LIN {X -0.074,Y -440.123,Z 231.770,A 0.000,B 0.000,C 90.000,E1 153.973} C_DIS
LIN {X 0.244,Y -443.570,Z 231.757,A 0.000,B 0.000,C 90.000,E1 151.307} C_DIS
LIN {X -0.099,Y -447.476,Z 231.744,A 0.000,B 0.000,C 90.000,E1 148.742} C_DIS
LIN {X -0.036,Y -450.606,Z 231.734,A 0.000,B 0.000,C 90.000,E1 146.786} C_DIS
LIN {X -0.031,Y -453.961,Z 231.724,A 0.000,B 0.000,C 90.000,E1 144.848} C_DIS
LIN {X -0.148,Y -456.732,Z 231.716,A 0.000,B 0.000,C 90.000,E1 143.256} C_DIS
LIN {X 0.157,Y -459.197,Z 231.708,A 0.000,B 0.000,C 90.000,E1 141.618} C_DIS
LIN {X -0.219,Y -461.363,Z 231.700,A 0.000,B 0.000,C 90.000,E1 140.070} C_DIS
LIN {X -0.002,Y -462.909,Z 231.694,A 0.000,B 0.000,C 90.000,E1 138.771} C_DIS
LIN {X -0.018,Y -464.342,Z 231.686,A 0.000,B 0.000,C 90.000,E1 137.187} C_DIS
LIN {X 0.219,Y -465.215,Z 231.680,A 0.000,B 0.000,C 90.000,E1 135.891} C_DIS
LIN {X -0.247,Y -465.696,Z 231.675,A 0.000,B 0.000,C 90.000,E1 135.000} C_DIS
LIN {X 0.017,Y -465.978,Z 231.669,A 0.000,B 0.000,C 90.000,E1 133.704} C_DIS
LIN {X -0.105,Y -465.940,Z 231.664,A 0.000,B 0.000,C 90.000,E1 132.771} C_DIS
LIN {X -0.166,Y -465.456,Z 231.657,A 0.000,B 0.000,C 90.000,E1 131.515} C_DIS
LIN {X -0.138,Y -464.609,Z 231.650,A 0.000,B 0.000,C 90.000,E1 129.930} C_DIS
LIN {X 0.071,Y -464.004,Z 231.645,A 0.000,B 0.000,C 90.000,E1 128.955} C_DIS
LIN {X 0.099,Y -462.931,Z 231.639,A 0.000,B 0.000,C 90.000,E1 127.684} C_DIS
LIN {X 0.027,Y -461.600,Z 231.632,A 0.000,B 0.000,C 90.000,E1 126.423} C_DIS
LIN {X 0.014,Y -460.384,Z 231.627,A 0.000,B 0.000,C 90.000,E1 125.471} C_DIS
LIN {X 0.112,Y -458.220,Z 231.619,A 0.000,B 0.000,C 90.000,E1 123.865} C_DIS
LIN {X -0.088,Y -455.689,Z 231.611,A 0.000,B 0.000,C 90.000,E1 122.291} C_DIS
LIN {X -0.055,Y -453.556,Z 231.605,A 0.000,B 0.000,C 90.000,E1 121.003} C_DIS
LIN {X -0.065,Y -451.335,Z 231.599,A 0.000,B 0.000,C 90.000,E1 119.716} C_DIS
LIN {X -0.010,Y -447.845,Z 231.589,A 0.000,B 0.000,C 90.000,E1 117.769} C_DIS
LIN {X -0.234,Y -444.436,Z 231.579,A 0.000,B 0.000,C 90.000,E1 115.848} C_DIS
LIN {X 0.063,Y -443.558,Z 231.577,A 0.000,B 0.000,C 90.000,E1 115.335} C_DIS
LIN {X 0.024,Y -443.550,Z 231.577,A 0.000,B 0.000,C 90.000,E1 115.335} C_DIS
LIN {X -0.070,Y -444.990,Z 231.574,A 0.000,B 0.000,C 90.000,E1 114.847} C_DIS
LIN {X 0.206,Y -454.125,Z 231.555,A 0.000,B 0.000,C 90.000,E1 110.918} C_DIS
LIN {X -0.107,Y -456.781,Z 231.550,A 0.000,B 0.000,C 90.000,E1 109.993} C_DIS
LIN {X 0.225,Y -457.541,Z 231.548,A 0.000,B 0.000,C 90.000,E1 109.631} C_DIS
LIN {X -0.136,Y -466.232,Z 231.528,A 0.000,B 0.000,C 90.000,E1 105.536} C_DIS
LIN {X -0.085,Y -467.792,Z 231.524,A 0.000,B 0.000,C 90.000,E1 104.898} C_DIS
LIN {X -0.114,Y -475.999,Z 231.501,A 0.000,B 0.000,C 90.000,E1 100.197} C_DIS
LIN {X 0.036,Y -476.693,Z 231.498,A 0.000,B 0.000,C 90.000,E1 99.557} C_DIS
LIN {X 0.160,Y -481.938,Z 231.478,A 0.000,B 0.000,C 90.000,E1 95.511} C_DIS
LIN {X 0.008,Y -482.209,Z 231.476,A 0.000,B 0.000,C 90.000,E1 95.220} C_DIS
LIN {X -0.054,Y -485.406,Z 231.455,A 0.000,B 0.000,C 90.000,E1 90.917} C_DIS
LIN {X -0.228,Y -485.528,Z 231.453,A 0.000,B 0.000,C 90.000,E1 90.630} C_DIS
LIN {X -0.021,Y -486.366,Z 231.433,A 0.000,B 0.000,C 90.000,E1 86.617} C_DIS
LIN {X -0.196,Y -486.368,Z 231.432,A 0.000,B 0.000,C 90.000,E1 86.331} C_DIS
LIN {X 0.138,Y -485.674,Z 231.425,A 0.000,B 0.000,C 90.000,E1 85.065} C_DIS
LIN {X -0.172,Y -484.691,Z 231.409,A 0.000,B 0.000,C 90.000,E1 81.724} C_DIS
LIN {X 0.174,Y -484.487,Z 231.407,A 0.000,B 0.000,C 90.000,E1 81.376} C_DIS
LIN {X 0.178,Y -480.662,Z 231.385,A 0.000,B 0.000,C 90.000,E1 77.061} C_DIS
LIN {X 0.144,Y -480.414,Z 231.384,A 0.000,B 0.000,C 90.000,E1 76.756} C_DIS
LIN {X -0.084,Y -474.193,Z 231.361,A 0.000,B 0.000,C 90.000,E1 72.127} C_DIS
LIN {X -0.150,Y -473.017,Z 231.357,A 0.000,B 0.000,C 90.000,E1 71.511} C_DIS
LIN {X -0.050,Y -465.699,Z 231.335,A 0.000,B 0.000,C 90.000,E1 67.102} C_DIS
LIN {X 0.008,Y -459.410,Z 231.321,A 0.000,B 0.000,C 90.000,E1 64.152} C_DIS
LIN {X -0.032,Y -459.417,Z 231.321,A 0.000,B 0.000,C 90.000,E1 64.152} C_DIS
LIN {X -0.197,Y -461.625,Z 231.317,A 0.000,B 0.000,C 90.000,E1 63.384} C_DIS
LIN {X -0.034,Y -464.697,Z 231.312,A 0.000,B 0.000,C 90.000,E1 62.410} C_DIS
LIN {X 0.169,Y -467.308,Z 231.307,A 0.000,B 0.000,C 90.000,E1 61.435} C_DIS
LIN {X -0.164,Y -468.856,Z 231.304,A 0.000,B 0.000,C 90.000,E1 60.845} C_DIS
LIN {X -0.007,Y -469.418,Z 231.303,A 0.000,B 0.000,C 90.000,E1 60.511} C_DIS
LIN {X -0.157,Y -470.244,Z 231.299,A 0.000,B 0.000,C 90.000,E1 59.744} C_DIS
LIN {X 0.008,Y -471.991,Z 231.296,A 0.000,B 0.000,C 90.000,E1 59.253} C_DIS
LIN {X -0.065,Y -473.436,Z 231.295,A 0.000,B 0.000,C 90.000,E1 58.948} C_DIS
LIN {X 0.111,Y -474.609,Z 231.293,A 0.000,B 0.000,C 90.000,E1 58.614} C_DIS
LIN {X 0.070,Y -476.278,Z 231.290,A 0.000,B 0.000,C 90.000,E1 57.995} C_DIS
LIN {X -0.146,Y -477.003,Z 231.288,A 0.000,B 0.000,C 90.000,E1 57.709} C_DIS
LIN {X 0.046,Y -477.537,Z 231.287,A 0.000,B 0.000,C 90.000,E1 57.375} C_DIS
LIN {X 0.007,Y -477.986,Z 231.285,A 0.000,B 0.000,C 90.000,E1 56.914} C_DIS
LIN {X -0.071,Y -480.360,Z 231.281,A 0.000,B 0.000,C 90.000,E1 56.294} C_DIS
LIN {X 0.129,Y -481.734,Z 231.280,A 0.000,B 0.000,C 90.000,E1 55.960} C_DIS
LIN {X -0.063,Y -482.676,Z 231.278,A 0.000,B 0.000,C 90.000,E1 55.674} C_DIS
LIN {X -0.253,Y -483.355,Z 231.277,A 0.000,B 0.000,C 90.000,E1 55.388} C_DIS
LIN {X -0.041,Y -483.816,Z 231.275,A 0.000,B 0.000,C 90.000,E1 55.055} C_DIS
LIN {X -0.223,Y -483.883,Z 231.274,A 0.000,B 0.000,C 90.000,E1 54.769} C_DIS
LIN {X -0.173,Y -483.679,Z 231.273,A 0.000,B 0.000,C 90.000,E1 54.609} C_DIS
LIN {X 0.180,Y -483.698,Z 231.273,A 0.000,B 0.000,C 90.000,E1 54.562} C_DIS
LIN {X 0.272,Y -484.576,Z 231.272,A 0.000,B 0.000,C 90.000,E1 54.402} C_DIS
LIN {X -0.082,Y -486.780,Z 231.269,A 0.000,B 0.000,C 90.000,E1 53.829} C_DIS
LIN {X 0.138,Y -487.584,Z 231.268,A 0.000,B 0.000,C 90.000,E1 53.497} C_DIS
LIN {X -0.032,Y -488.131,Z 231.266,A 0.000,B 0.000,C 90.000,E1 53.210} C_DIS
LIN {X -0.199,Y -488.277,Z 231.265,A 0.000,B 0.000,C 90.000,E1 52.924} C_DIS
LIN {X 0.192,Y -487.980,Z 231.262,A 0.000,B 0.000,C 90.000,E1 52.477} C_DIS
LIN {X 0.151,Y -487.990,Z 231.262,A 0.000,B 0.000,C 90.000,E1 52.477} C_DIS
LIN {X 0.157,Y -489.294,Z 231.261,A 0.000,B 0.000,C 90.000,E1 52.271} C_DIS
LIN {X -0.007,Y -490.426,Z 231.260,A 0.000,B 0.000,C 90.000,E1 51.984} C_DIS
LIN {X -0.169,Y -491.097,Z 231.258,A 0.000,B 0.000,C 90.000,E1 51.698} C_DIS
LIN {X -0.022,Y -491.509,Z 231.257,A 0.000,B 0.000,C 90.000,E1 51.376} C_DIS
LIN {X -0.317,Y -492.691,Z 231.254,A 0.000,B 0.000,C 90.000,E1 50.803} C_DIS
LIN {X 0.071,Y -493.673,Z 231.251,A 0.000,B 0.000,C 90.000,E1 50.150} C_DIS
LIN {X 0.237,Y -493.877,Z 231.249,A 0.000,B 0.000,C 90.000,E1 49.828} C_DIS
LIN {X 0.004,Y -493.736,Z 231.249,A 0.000,B 0.000,C 90.000,E1 49.703} C_DIS
LIN {X 0.088,Y -494.275,Z 231.248,A 0.000,B 0.000,C 90.000,E1 49.542} C_DIS
LIN {X -0.062,Y -495.108,Z 231.246,A 0.000,B 0.000,C 90.000,E1 49.256} C_DIS
LIN {X 0.112,Y -495.730,Z 231.245,A 0.000,B 0.000,C 90.000,E1 48.933} C_DIS
LIN {X -0.036,Y -496.097,Z 231.243,A 0.000,B 0.000,C 90.000,E1 48.647} C_DIS
LIN {X 0.145,Y -495.824,Z 231.242,A 0.000,B 0.000,C 90.000,E1 48.324} C_DIS
LIN {X 0.279,Y -495.320,Z 231.241,A 0.000,B 0.000,C 90.000,E1 48.162} C_DIS
LIN {X 0.237,Y -495.320,Z 231.241,A 0.000,B 0.000,C 90.000,E1 48.162} C_DIS
LIN {X -0.001,Y -495.841,Z 231.240,A 0.000,B 0.000,C 90.000,E1 48.038} C_DIS
LIN {X 0.001,Y -497.005,Z 231.237,A 0.000,B 0.000,C 90.000,E1 47.433} C_DIS
LIN {X -0.103,Y -498.434,Z 231.233,A 0.000,B 0.000,C 90.000,E1 46.539} C_DIS
LIN {X 0.093,Y -498.808,Z 231.231,A 0.000,B 0.000,C 90.000,E1 46.215} C_DIS
LIN {X 0.292,Y -498.427,Z 231.230,A 0.000,B 0.000,C 90.000,E1 45.891} C_DIS
LIN {X -0.313,Y -497.786,Z 231.229,A 0.000,B 0.000,C 90.000,E1 45.810} C_DIS
LIN {X 0.002,Y -497.788,Z 231.229,A 0.000,B 0.000,C 90.000,E1 45.769} C_DIS
LIN {X -0.213,Y -498.693,Z 231.228,A 0.000,B 0.000,C 90.000,E1 45.648} C_DIS
LIN {X -0.015,Y -499.458,Z 231.227,A 0.000,B 0.000,C 90.000,E1 45.324} C_DIS
LIN {X 0.186,Y -499.495,Z 231.225,A 0.000,B 0.000,C 90.000,E1 45.000} C_DIS
LIN {X 0.143,Y -498.484,Z 231.223,A 0.000,B 0.000,C 90.000,E1 44.676} C_DIS
LIN {X 0.102,Y -498.455,Z 231.223,A 0.000,B 0.000,C 90.000,E1 44.676} C_DIS
LIN {X -0.215,Y -498.923,Z 231.223,A 0.000,B 0.000,C 90.000,E1 44.595} C_DIS
LIN {X -0.114,Y -499.227,Z 231.222,A 0.000,B 0.000,C 90.000,E1 44.433} C_DIS
LIN {X 0.087,Y -499.387,Z 231.221,A 0.000,B 0.000,C 90.000,E1 44.109} C_DIS
LIN {X 0.206,Y -498.913,Z 231.219,A 0.000,B 0.000,C 90.000,E1 43.785} C_DIS
LIN {X 0.165,Y -498.902,Z 231.219,A 0.000,B 0.000,C 90.000,E1 43.785} C_DIS
LIN {X 0.045,Y -499.551,Z 231.218,A 0.000,B 0.000,C 90.000,E1 43.662} C_DIS
LIN {X -0.216,Y -499.927,Z 231.218,A 0.000,B 0.000,C 90.000,E1 43.542} C_DIS
LIN {X -0.014,Y -500.088,Z 231.216,A 0.000,B 0.000,C 90.000,E1 43.218} C_DIS
LIN {X -0.152,Y -499.878,Z 231.215,A 0.000,B 0.000,C 90.000,E1 42.933} C_DIS
LIN {X -0.255,Y -499.278,Z 231.214,A 0.000,B 0.000,C 90.000,E1 42.771} C_DIS
LIN {X -0.296,Y -499.296,Z 231.214,A 0.000,B 0.000,C 90.000,E1 42.771} C_DIS
LIN {X 0.052,Y -499.752,Z 231.213,A 0.000,B 0.000,C 90.000,E1 42.609} C_DIS
LIN {X -0.085,Y -500.114,Z 231.212,A 0.000,B 0.000,C 90.000,E1 42.324} C_DIS
LIN {X 0.117,Y -499.916,Z 231.210,A 0.000,B 0.000,C 90.000,E1 42.000} C_DIS
LIN {X 0.218,Y -499.485,Z 231.209,A 0.000,B 0.000,C 90.000,E1 41.838} C_DIS
LIN {X -0.263,Y -498.757,Z 231.209,A 0.000,B 0.000,C 90.000,E1 41.757} C_DIS
LIN {X -0.305,Y -498.741,Z 231.209,A 0.000,B 0.000,C 90.000,E1 41.757} C_DIS
LIN {X 0.183,Y -499.759,Z 231.207,A 0.000,B 0.000,C 90.000,E1 41.391} C_DIS
LIN {X -0.328,Y -499.706,Z 231.206,A 0.000,B 0.000,C 90.000,E1 41.148} C_DIS
LIN {X 0.133,Y -498.220,Z 231.204,A 0.000,B 0.000,C 90.000,E1 40.701} C_DIS
LIN {X 0.092,Y -498.225,Z 231.204,A 0.000,B 0.000,C 90.000,E1 40.701} C_DIS
LIN {X -0.261,Y -498.803,Z 231.203,A 0.000,B 0.000,C 90.000,E1 40.539} C_DIS
LIN {X -0.071,Y -499.213,Z 231.201,A 0.000,B 0.000,C 90.000,E1 40.216} C_DIS
LIN {X -0.017,Y -498.068,Z 231.194,A 0.000,B 0.000,C 90.000,E1 38.705} C_DIS
LIN {X 0.032,Y -497.387,Z 231.191,A 0.000,B 0.000,C 90.000,E1 38.096} C_DIS
LIN {X -0.098,Y -496.913,Z 231.189,A 0.000,B 0.000,C 90.000,E1 37.810} C_DIS
LIN {X -0.231,Y -496.627,Z 231.187,A 0.000,B 0.000,C 90.000,E1 37.523} C_DIS
LIN {X -0.217,Y -494.491,Z 231.180,A 0.000,B 0.000,C 90.000,E1 36.011} C_DIS
LIN {X -0.132,Y -491.985,Z 231.172,A 0.000,B 0.000,C 90.000,E1 34.485} C_DIS
LIN {X -0.184,Y -490.288,Z 231.168,A 0.000,B 0.000,C 90.000,E1 33.579} C_DIS
LIN {X -0.094,Y -489.022,Z 231.165,A 0.000,B 0.000,C 90.000,E1 32.959} C_DIS
LIN {X 0.052,Y -487.027,Z 231.159,A 0.000,B 0.000,C 90.000,E1 31.720} C_DIS
LIN {X 0.091,Y -485.337,Z 231.154,A 0.000,B 0.000,C 90.000,E1 30.797} C_DIS
LIN {X -0.112,Y -484.619,Z 231.151,A 0.000,B 0.000,C 90.000,E1 30.207} C_DIS
LIN {X 0.128,Y -482.896,Z 231.145,A 0.000,B 0.000,C 90.000,E1 28.949} C_DIS
LIN {X -0.076,Y -482.340,Z 231.143,A 0.000,B 0.000,C 90.000,E1 28.665} C_DIS
LIN {X -0.091,Y -482.066,Z 231.142,A 0.000,B 0.000,C 90.000,E1 28.359} C_DIS
LIN {X -0.214,Y -478.844,Z 231.126,A 0.000,B 0.000,C 90.000,E1 25.283} C_DIS
LIN {X -0.055,Y -478.231,Z 231.122,A 0.000,B 0.000,C 90.000,E1 24.335} C_DIS
LIN {X 0.041,Y -476.845,Z 231.112,A 0.000,B 0.000,C 90.000,E1 22.461} C_DIS
LIN {X -0.105,Y -475.134,Z 231.101,A 0.000,B 0.000,C 90.000,E1 20.301} C_DIS
LIN {X 0.101,Y -474.287,Z 231.097,A 0.000,B 0.000,C 90.000,E1 19.341} C_DIS
LIN {X 0.041,Y -473.953,Z 231.094,A 0.000,B 0.000,C 90.000,E1 18.725} C_DIS
LIN {X 0.021,Y -472.799,Z 231.086,A 0.000,B 0.000,C 90.000,E1 17.166} C_DIS
LIN {X -0.066,Y -472.038,Z 231.083,A 0.000,B 0.000,C 90.000,E1 16.551} C_DIS
LIN {X -0.077,Y -471.535,Z 231.076,A 0.000,B 0.000,C 90.000,E1 15.300} C_DIS
LIN {X -0.182,Y -470.205,Z 231.065,A 0.000,B 0.000,C 90.000,E1 13.119} C_DIS
LIN {X 0.217,Y -469.233,Z 231.056,A 0.000,B 0.000,C 90.000,E1 11.186} C_DIS
LIN {X 0.228,Y -468.732,Z 231.048,A 0.000,B 0.000,C 90.000,E1 9.613} C_DIS
LIN {X -0.037,Y -468.156,Z 231.039,A 0.000,B 0.000,C 90.000,E1 7.757} C_DIS
LIN {X 0.064,Y -467.837,Z 231.032,A 0.000,B 0.000,C 90.000,E1 6.486} C_DIS
LIN {X 0.156,Y -467.773,Z 231.014,A 0.000,B 0.000,C 90.000,E1 2.694} C_DIS
LIN {X -0.017,Y -469.620,Z 231.000,A 0.000,B 0.000,C 90.000,E1 357.593} C_DIS
LIN {X -0.162,Y -471.139,Z 231.000,A 0.000,B 0.000,C 90.000,E1 355.412} C_DIS
LIN {X -0.107,Y -475.620,Z 231.000,A 0.000,B 0.000,C 90.000,E1 351.027} C_DIS
LIN {X 0.191,Y -477.529,Z 231.000,A 0.000,B 0.000,C 90.000,E1 349.746} C_DIS
LIN {X -0.094,Y -480.696,Z 231.000,A 0.000,B 0.000,C 90.000,E1 348.229} C_DIS
LIN {X -0.276,Y -488.714,Z 231.000,A 0.000,B 0.000,C 90.000,E1 345.172} C_DIS
LIN {X -0.079,Y -494.405,Z 231.000,A 0.000,B 0.000,C 90.000,E1 343.015} C_DIS
LIN {X -0.087,Y -503.824,Z 231.000,A 0.000,B 0.000,C 90.000,E1 339.699} C_DIS
LIN {X -0.251,Y -513.500,Z 231.000,A 0.000,B 0.000,C 90.000,E1 336.741} C_DIS
LIN {X -0.229,Y -519.706,Z 231.000,A 0.000,B 0.000,C 90.000,E1 334.973} C_DIS
LIN {X -0.069,Y -526.045,Z 231.000,A 0.000,B 0.000,C 90.000,E1 333.204} C_DIS
LIN {X 0.245,Y -532.623,Z 231.000,A 0.000,B 0.000,C 90.000,E1 331.435} C_DIS
LIN {X 0.265,Y -538.025,Z 231.000,A 0.000,B 0.000,C 90.000,E1 329.999} C_DIS
LIN {X -0.096,Y -543.297,Z 231.000,A 0.000,B 0.000,C 90.000,E1 328.614} C_DIS
LIN {X -0.053,Y -549.622,Z 231.000,A 0.000,B 0.000,C 90.000,E1 326.914} C_DIS
LIN {X -0.261,Y -557.113,Z 231.000,A 0.000,B 0.000,C 90.000,E1 324.975} C_DIS
LIN {X 0.171,Y -562.435,Z 231.000,A 0.000,B 0.000,C 90.000,E1 323.543} C_DIS
LIN {X 0.142,Y -565.560,Z 231.000,A 0.000,B 0.000,C 90.000,E1 322.718} C_DIS
LIN {X -0.041,Y -571.531,Z 231.000,A 0.000,B 0.000,C 90.000,E1 321.090} C_DIS
LIN {X 0.030,Y -581.801,Z 231.000,A 0.000,B 0.000,C 90.000,E1 318.366} C_DIS
LIN {X 0.089,Y -585.027,Z 231.000,A 0.000,B 0.000,C 90.000,E1 317.553} C_DIS
LIN {X 0.145,Y -588.340,Z 231.000,A 0.000,B 0.000,C 90.000,E1 316.743} C_DIS
LIN {X 0.075,Y -590.482,Z 231.000,A 0.000,B 0.000,C 90.000,E1 316.215} C_DIS
LIN {X -0.274,Y -595.173,Z 231.000,A 0.000,B 0.000,C 90.000,E1 314.919} C_DIS
LIN {X 0.297,Y -598.942,Z 231.000,A 0.000,B 0.000,C 90.000,E1 313.542} C_DIS
LIN {X 0.089,Y -600.943,Z 231.000,A 0.000,B 0.000,C 90.000,E1 312.771} C_DIS
LIN {X -0.305,Y -603.007,Z 231.000,A 0.000,B 0.000,C 90.000,E1 311.757} C_DIS
LIN {X -0.220,Y -604.627,Z 231.000,A 0.000,B 0.000,C 90.000,E1 310.701} C_DIS
LIN {X -0.055,Y -606.637,Z 231.000,A 0.000,B 0.000,C 90.000,E1 309.116} C_DIS
LIN {X -0.308,Y -607.723,Z 231.000,A 0.000,B 0.000,C 90.000,E1 308.096} C_DIS
LIN {X -0.062,Y -608.527,Z 231.000,A 0.000,B 0.000,C 90.000,E1 307.030} C_DIS
LIN {X -0.292,Y -609.123,Z 231.000,A 0.000,B 0.000,C 90.000,E1 306.011} C_DIS
LIN {X -0.029,Y -609.527,Z 231.000,A 0.000,B 0.000,C 90.000,E1 304.945} C_DIS
LIN {X -0.111,Y -609.714,Z 231.000,A 0.000,B 0.000,C 90.000,E1 303.913} C_DIS
LIN {X -0.190,Y -609.416,Z 231.000,A 0.000,B 0.000,C 90.000,E1 302.880} C_DIS
LIN {X 0.025,Y -609.165,Z 231.000,A 0.000,B 0.000,C 90.000,E1 302.339} C_DIS
LIN {X -0.387,Y -608.149,Z 231.000,A 0.000,B 0.000,C 90.000,E1 301.337} C_DIS
LIN {X -0.232,Y -607.105,Z 231.000,A 0.000,B 0.000,C 90.000,E1 300.541} C_DIS
LIN {X 0.156,Y -605.445,Z 231.000,A 0.000,B 0.000,C 90.000,E1 299.461} C_DIS
LIN {X -0.074,Y -603.446,Z 231.000,A 0.000,B 0.000,C 90.000,E1 298.437} C_DIS
LIN {X -0.041,Y -601.174,Z 231.000,A 0.000,B 0.000,C 90.000,E1 297.385} C_DIS
LIN {X 0.144,Y -598.015,Z 231.000,A 0.000,B 0.000,C 90.000,E1 296.052} C_DIS
LIN {X -0.261,Y -594.859,Z 231.000,A 0.000,B 0.000,C 90.000,E1 294.771} C_DIS
LIN {X -0.092,Y -592.135,Z 231.000,A 0.000,B 0.000,C 90.000,E1 293.695} C_DIS
LIN {X 0.209,Y -587.297,Z 231.000,A 0.000,B 0.000,C 90.000,E1 291.535} C_DIS
LIN {X 0.025,Y -582.165,Z 231.000,A 0.000,B 0.000,C 90.000,E1 289.141} C_DIS
LIN {X -0.184,Y -578.311,Z 231.000,A 0.000,B 0.000,C 90.000,E1 287.275} C_DIS
LIN {X -0.094,Y -574.648,Z 231.000,A 0.000,B 0.000,C 90.000,E1 285.371} C_DIS
LIN {X 0.091,Y -570.891,Z 231.000,A 0.000,B 0.000,C 90.000,E1 283.175} C_DIS
LIN {X 0.078,Y -567.291,Z 231.000,A 0.000,B 0.000,C 90.000,E1 280.715} C_DIS
LIN {X -0.023,Y -565.032,Z 231.000,A 0.000,B 0.000,C 90.000,E1 278.803} C_DIS
LIN {X 0.194,Y -561.526,Z 231.000,A 0.000,B 0.000,C 90.000,E1 274.645} C_DIS
LIN {X -0.002,Y -560.683,Z 231.000,A 0.000,B 0.000,C 90.000,E1 270.516} C_DIS
LIN {X 0.106,Y -561.025,Z 231.000,A 0.000,B 0.000,C 90.000,E1 268.568} C_DIS
LIN {X 0.202,Y -565.510,Z 231.000,A 0.000,B 0.000,C 90.000,E1 262.761} C_DIS
LIN {X 0.182,Y -568.294,Z 231.000,A 0.000,B 0.000,C 90.000,E1 260.566} C_DIS
LIN {X -0.140,Y -571.593,Z 231.000,A 0.000,B 0.000,C 90.000,E1 258.409} C_DIS
LIN {X -0.164,Y -573.802,Z 231.000,A 0.000,B 0.000,C 90.000,E1 257.048} C_DIS
LIN {X -0.273,Y -575.852,Z 231.000,A 0.000,B 0.000,C 90.000,E1 255.700} C_DIS
LIN {X -0.214,Y -577.769,Z 231.000,A 0.000,B 0.000,C 90.000,E1 254.338} C_DIS
LIN {X -0.172,Y -579.165,Z 231.000,A 0.000,B 0.000,C 90.000,E1 253.251} C_DIS
LIN {X -0.277,Y -580.278,Z 231.000,A 0.000,B 0.000,C 90.000,E1 252.181} C_DIS
LIN {X -0.237,Y -580.622,Z 231.000,A 0.000,B 0.000,C 90.000,E1 251.638} C_DIS
LIN {X 0.197,Y -580.838,Z 231.000,A 0.000,B 0.000,C 90.000,E1 250.786} C_DIS
LIN {X -0.261,Y -580.913,Z 231.000,A 0.000,B 0.000,C 90.000,E1 249.752} C_DIS
LIN {X 0.029,Y -580.630,Z 231.000,A 0.000,B 0.000,C 90.000,E1 248.646} C_DIS
LIN {X -0.330,Y -580.541,Z 231.000,A 0.000,B 0.000,C 90.000,E1 248.411} C_DIS
LIN {X -0.200,Y -579.237,Z 231.000,A 0.000,B 0.000,C 90.000,E1 247.050} C_DIS
LIN {X 0.133,Y -577.281,Z 231.000,A 0.000,B 0.000,C 90.000,E1 245.665} C_DIS
LIN {X 0.213,Y -575.764,Z 231.000,A 0.000,B 0.000,C 90.000,E1 244.845} C_DIS
LIN {X -0.039,Y -572.673,Z 231.000,A 0.000,B 0.000,C 90.000,E1 243.512} C_DIS
LIN {X 0.081,Y -569.984,Z 231.000,A 0.000,B 0.000,C 90.000,E1 242.410} C_DIS
LIN {X 0.069,Y -567.822,Z 231.000,A 0.000,B 0.000,C 90.000,E1 241.591} C_DIS
LIN {X -0.198,Y -565.488,Z 231.000,A 0.000,B 0.000,C 90.000,E1 240.795} C_DIS
LIN {X -0.019,Y -560.734,Z 231.000,A 0.000,B 0.000,C 90.000,E1 239.125} C_DIS
LIN {X -0.020,Y -556.515,Z 231.000,A 0.000,B 0.000,C 90.000,E1 237.740} C_DIS
LIN {X 0.031,Y -552.250,Z 231.000,A 0.000,B 0.000,C 90.000,E1 236.342} C_DIS
LIN {X -0.035,Y -548.591,Z 231.000,A 0.000,B 0.000,C 90.000,E1 235.229} C_DIS
LIN {X -0.073,Y -543.215,Z 231.000,A 0.000,B 0.000,C 90.000,E1 233.543} C_DIS
LIN {X 0.049,Y -539.595,Z 231.000,A 0.000,B 0.000,C 90.000,E1 232.396} C_DIS
LIN {X 0.118,Y -535.201,Z 231.000,A 0.000,B 0.000,C 90.000,E1 230.964} C_DIS
LIN {X 0.036,Y -531.590,Z 231.000,A 0.000,B 0.000,C 90.000,E1 229.828} C_DIS
LIN {X -0.123,Y -526.808,Z 231.000,A 0.000,B 0.000,C 90.000,E1 228.405} C_DIS
LIN {X -0.278,Y -524.063,Z 231.000,A 0.000,B 0.000,C 90.000,E1 227.553} C_DIS
LIN {X -0.319,Y -518.248,Z 231.000,A 0.000,B 0.000,C 90.000,E1 225.810} C_DIS
LIN {X 0.069,Y -514.580,Z 231.000,A 0.000,B 0.000,C 90.000,E1 224.595} C_DIS
LIN {X 0.137,Y -511.656,Z 231.000,A 0.000,B 0.000,C 90.000,E1 223.704} C_DIS
LIN {X -0.038,Y -507.055,Z 231.000,A 0.000,B 0.000,C 90.000,E1 222.243} C_DIS
LIN {X -0.120,Y -499.087,Z 231.000,A 0.000,B 0.000,C 90.000,E1 219.564} C_DIS
LIN {X 0.096,Y -493.914,Z 231.000,A 0.000,B 0.000,C 90.000,E1 217.729} C_DIS
LIN {X -0.109,Y -488.935,Z 231.000,A 0.000,B 0.000,C 90.000,E1 215.931} C_DIS
LIN {X 0.088,Y -483.787,Z 231.000,A 0.000,B 0.000,C 90.000,E1 214.072} C_DIS
LIN {X -0.057,Y -481.287,Z 231.000,A 0.000,B 0.000,C 90.000,E1 213.166} C_DIS
LIN {X 0.095,Y -474.345,Z 231.000,A 0.000,B 0.000,C 90.000,E1 210.669} C_DIS
LIN {X -0.200,Y -465.869,Z 231.000,A 0.000,B 0.000,C 90.000,E1 207.257} C_DIS
LIN {X -0.220,Y -458.796,Z 231.000,A 0.000,B 0.000,C 90.000,E1 203.770} C_DIS
LIN {X -0.136,Y -451.228,Z 231.000,A 0.000,B 0.000,C 90.000,E1 199.268} C_DIS
LIN {X -0.116,Y -447.580,Z 231.000,A 0.000,B 0.000,C 90.000,E1 196.677} C_DIS
LIN {X -0.033,Y -444.252,Z 231.000,A 0.000,B 0.000,C 90.000,E1 194.064} C_DIS
LIN {X 0.121,Y -442.239,Z 231.000,A 0.000,B 0.000,C 90.000,E1 192.411} C_DIS
LIN {X -0.228,Y -439.819,Z 231.000,A 0.000,B 0.000,C 90.000,E1 190.489} C_DIS
LIN {X -0.050,Y -437.322,Z 231.000,A 0.000,B 0.000,C 90.000,E1 188.163} C_DIS
LIN {X -0.073,Y -435.000,Z 231.000,A 0.000,B 0.000,C 90.000,E1 185.853} C_DIS
LIN {X 0.192,Y -433.100,Z 231.000,A 0.000,B 0.000,C 90.000,E1 183.498} C_DIS
LIN {X -0.136,Y -431.588,Z 231.000,A 0.000,B 0.000,C 90.000,E1 181.547} C_DIS
LIN {X 0.001,Y -428.996,Z 231.000,A 0.000,B 0.000,C 90.000,E1 177.192} C_DIS
LIN {X 0.201,Y -428.276,Z 231.000,A 0.000,B 0.000,C 90.000,E1 174.489} C_DIS
LIN {X -0.018,Y -428.328,Z 231.000,A 0.000,B 0.000,C 90.000,E1 173.514} C_DIS
LIN {X -0.107,Y -428.536,Z 231.000,A 0.000,B 0.000,C 90.000,E1 170.849} C_DIS
LIN {X 0.100,Y -428.906,Z 231.000,A 0.000,B 0.000,C 90.000,E1 168.814} C_DIS
LIN {X -0.029,Y -429.592,Z 231.000,A 0.000,B 0.000,C 90.000,E1 166.825} C_DIS
LIN {X 0.055,Y -430.492,Z 231.000,A 0.000,B 0.000,C 90.000,E1 164.810} C_DIS
LIN {X 0.166,Y -431.099,Z 231.000,A 0.000,B 0.000,C 90.000,E1 163.795} C_DIS
LIN {X -0.152,Y -431.375,Z 231.000,A 0.000,B 0.000,C 90.000,E1 163.504} C_DIS
LIN {X -0.066,Y -433.126,Z 231.000,A 0.000,B 0.000,C 90.000,E1 160.496} C_DIS
LIN {X -0.201,Y -433.876,Z 231.000,A 0.000,B 0.000,C 90.000,E1 159.518} C_DIS
LIN {X -0.052,Y -436.169,Z 231.000,A 0.000,B 0.000,C 90.000,E1 156.847} C_DIS
LIN {X -0.043,Y -439.056,Z 231.000,A 0.000,B 0.000,C 90.000,E1 154.204} C_DIS
LIN {X 0.048,Y -442.464,Z 231.000,A 0.000,B 0.000,C 90.000,E1 151.563} C_DIS
LIN {X 0.058,Y -446.337,Z 231.000,A 0.000,B 0.000,C 90.000,E1 148.948} C_DIS
LIN {X 0.094,Y -449.469,Z 231.000,A 0.000,B 0.000,C 90.000,E1 146.993} C_DIS
LIN {X -0.213,Y -453.348,Z 231.000,A 0.000,B 0.000,C 90.000,E1 144.769} C_DIS
LIN {X 0.026,Y -456.122,Z 231.000,A 0.000,B 0.000,C 90.000,E1 143.130} C_DIS
LIN {X -0.044,Y -458.604,Z 231.000,A 0.000,B 0.000,C 90.000,E1 141.537} C_DIS
LIN {X -0.167,Y -460.378,Z 231.000,A 0.000,B 0.000,C 90.000,E1 140.275} C_DIS
LIN {X -0.222,Y -462.328,Z 231.000,A 0.000,B 0.000,C 90.000,E1 138.690} C_DIS
LIN {X 0.011,Y -463.485,Z 231.000,A 0.000,B 0.000,C 90.000,E1 137.391} C_DIS
LIN {X -0.081,Y -464.386,Z 231.000,A 0.000,B 0.000,C 90.000,E1 136.134} C_DIS
LIN {X 0.163,Y -465.017,Z 231.000,A 0.000,B 0.000,C 90.000,E1 134.838} C_DIS
LIN {X -0.305,Y -465.282,Z 231.000,A 0.000,B 0.000,C 90.000,E1 133.947} C_DIS
LIN {X 0.285,Y -465.213,Z 231.000,A 0.000,B 0.000,C 90.000,E1 132.609} C_DIS
LIN {X -0.096,Y -464.728,Z 231.000,A 0.000,B 0.000,C 90.000,E1 131.391} C_DIS
LIN {X 0.173,Y -464.096,Z 231.000,A 0.000,B 0.000,C 90.000,E1 130.092} C_DIS
LIN {X 0.129,Y -463.276,Z 231.000,A 0.000,B 0.000,C 90.000,E1 128.830} C_DIS
LIN {X 0.183,Y -461.918,Z 231.000,A 0.000,B 0.000,C 90.000,E1 127.237} C_DIS
LIN {X -0.182,Y -460.478,Z 231.000,A 0.000,B 0.000,C 90.000,E1 126.011} C_DIS
LIN {X 0.027,Y -457.941,Z 231.000,A 0.000,B 0.000,C 90.000,E1 124.072} C_DIS
LIN {X 0.067,Y -455.447,Z 231.000,A 0.000,B 0.000,C 90.000,E1 122.467} C_DIS
LIN {X -0.146,Y -453.364,Z 231.000,A 0.000,B 0.000,C 90.000,E1 121.209} C_DIS
LIN {X -0.068,Y -450.561,Z 231.000,A 0.000,B 0.000,C 90.000,E1 119.589} C_DIS
LIN {X -0.100,Y -447.682,Z 231.000,A 0.000,B 0.000,C 90.000,E1 117.975} C_DIS
LIN {X -0.126,Y -444.272,Z 231.000,A 0.000,B 0.000,C 90.000,E1 116.027} C_DIS
LIN {X -0.143,Y -443.238,Z 231.000,A 0.000,B 0.000,C 90.000,E1 115.463} C_DIS
LIN {X -0.182,Y -443.246,Z 231.000,A 0.000,B 0.000,C 90.000,E1 115.463} C_DIS
LIN {X 0.031,Y -444.480,Z 231.000,A 0.000,B 0.000,C 90.000,E1 115.027} C_DIS
LIN {X -0.070,Y -445.942,Z 231.000,A 0.000,B 0.000,C 90.000,E1 114.387} C_DIS
LIN {X 0.066,Y -455.355,Z 231.000,A 0.000,B 0.000,C 90.000,E1 110.482} C_DIS
LIN {X -0.138,Y -457.153,Z 231.000,A 0.000,B 0.000,C 90.000,E1 109.866} C_DIS
LIN {X 0.158,Y -466.550,Z 231.000,A 0.000,B 0.000,C 90.000,E1 105.371} C_DIS
LIN {X -0.115,Y -467.999,Z 231.000,A 0.000,B 0.000,C 90.000,E1 104.773} C_DIS
LIN {X -0.152,Y -476.216,Z 231.000,A 0.000,B 0.000,C 90.000,E1 100.074} C_DIS
LIN {X 0.103,Y -482.115,Z 231.000,A 0.000,B 0.000,C 90.000,E1 95.391} C_DIS
LIN {X -0.148,Y -485.521,Z 231.000,A 0.000,B 0.000,C 90.000,E1 90.802} C_DIS
LIN {X -0.115,Y -486.381,Z 231.000,A 0.000,B 0.000,C 90.000,E1 86.502} C_DIS
LIN {X 0.194,Y -486.356,Z 231.000,A 0.000,B 0.000,C 90.000,E1 86.159} C_DIS
LIN {X -0.207,Y -484.675,Z 231.000,A 0.000,B 0.000,C 90.000,E1 81.602} C_DIS
LIN {X 0.162,Y -480.593,Z 231.000,A 0.000,B 0.000,C 90.000,E1 76.937} C_DIS
LIN {X -0.125,Y -479.688,Z 231.000,A 0.000,B 0.000,C 90.000,E1 76.353} C_DIS
LIN {X -0.092,Y -474.030,Z 231.000,A 0.000,B 0.000,C 90.000,E1 72.000} C_DIS
LIN {X -0.004,Y -465.950,Z 231.000,A 0.000,B 0.000,C 90.000,E1 67.283} C_DIS
LIN {X -0.061,Y -465.451,Z 231.000,A 0.000,B 0.000,C 90.000,E1 66.975} C_DIS
LIN {X -0.143,Y -459.228,Z 231.000,A 0.000,B 0.000,C 90.000,E1 64.076} C_DIS
LIN {X 0.230,Y -459.231,Z 231.000,A 0.000,B 0.000,C 90.000,E1 64.024} C_DIS
LIN {X 0.144,Y -462.994,Z 231.000,A 0.000,B 0.000,C 90.000,E1 62.820} C_DIS
LIN {X -0.225,Y -465.008,Z 231.000,A 0.000,B 0.000,C 90.000,E1 62.231} C_DIS
LIN {X -0.024,Y -467.554,Z 231.000,A 0.000,B 0.000,C 90.000,E1 61.257} C_DIS
LIN {X 0.125,Y -468.281,Z 231.000,A 0.000,B 0.000,C 90.000,E1 60.923} C_DIS
LIN {X 0.279,Y -468.858,Z 231.000,A 0.000,B 0.000,C 90.000,E1 60.589} C_DIS
LIN {X -0.043,Y -469.473,Z 231.000,A 0.000,B 0.000,C 90.000,E1 59.999} C_DIS
LIN {X -0.283,Y -469.598,Z 231.000,A 0.000,B 0.000,C 90.000,E1 59.871} C_DIS
LIN {X 0.119,Y -470.041,Z 231.000,A 0.000,B 0.000,C 90.000,E1 59.665} C_DIS
LIN {X -0.004,Y -471.928,Z 231.000,A 0.000,B 0.000,C 90.000,E1 59.203} C_DIS
LIN {X -0.258,Y -473.616,Z 231.000,A 0.000,B 0.000,C 90.000,E1 58.869} C_DIS
LIN {X 0.155,Y -474.204,Z 231.000,A 0.000,B 0.000,C 90.000,E1 58.663} C_DIS
LIN {X -0.136,Y -475.861,Z 231.000,A 0.000,B 0.000,C 90.000,E1 58.074} C_DIS
LIN {X 0.048,Y -476.558,Z 231.000,A 0.000,B 0.000,C 90.000,E1 57.740} C_DIS
LIN {X -0.166,Y -477.052,Z 231.000,A 0.000,B 0.000,C 90.000,E1 57.454} C_DIS
LIN {X 0.051,Y -477.508,Z 231.000,A 0.000,B 0.000,C 90.000,E1 56.962} C_DIS
LIN {X 0.173,Y -478.670,Z 231.000,A 0.000,B 0.000,C 90.000,E1 56.628} C_DIS
LIN {X 0.137,Y -480.536,Z 231.000,A 0.000,B 0.000,C 90.000,E1 56.167} C_DIS
LIN {X 0.171,Y -481.226,Z 231.000,A 0.000,B 0.000,C 90.000,E1 56.008} C_DIS
LIN {X -0.022,Y -482.310,Z 231.000,A 0.000,B 0.000,C 90.000,E1 55.722} C_DIS
LIN {X 0.187,Y -482.983,Z 231.000,A 0.000,B 0.000,C 90.000,E1 55.388} C_DIS
LIN {X 0.001,Y -483.425,Z 231.000,A 0.000,B 0.000,C 90.000,E1 55.102} C_DIS
LIN {X 0.213,Y -483.467,Z 231.000,A 0.000,B 0.000,C 90.000,E1 54.769} C_DIS
LIN {X -0.062,Y -483.148,Z 231.000,A 0.000,B 0.000,C 90.000,E1 54.609} C_DIS
LIN {X -0.102,Y -483.161,Z 231.000,A 0.000,B 0.000,C 90.000,E1 54.609} C_DIS
LIN {X 0.032,Y -483.942,Z 231.000,A 0.000,B 0.000,C 90.000,E1 54.482} C_DIS
LIN {X -0.149,Y -485.170,Z 231.000,A 0.000,B 0.000,C 90.000,E1 54.196} C_DIS
LIN {X 0.066,Y -486.272,Z 231.000,A 0.000,B 0.000,C 90.000,E1 53.863} C_DIS
LIN {X -0.110,Y -487.224,Z 231.000,A 0.000,B 0.000,C 90.000,E1 53.577} C_DIS
LIN {X 0.009,Y -487.767,Z 231.000,A 0.000,B 0.000,C 90.000,E1 53.256} C_DIS
LIN {X -0.157,Y -487.901,Z 231.000,A 0.000,B 0.000,C 90.000,E1 52.970} C_DIS
LIN {X 0.254,Y -487.582,Z 231.000,A 0.000,B 0.000,C 90.000,E1 52.477} C_DIS
LIN {X 0.213,Y -487.590,Z 231.000,A 0.000,B 0.000,C 90.000,E1 52.477} C_DIS
LIN {X -0.034,Y -489.510,Z 231.000,A 0.000,B 0.000,C 90.000,E1 52.190} C_DIS
LIN {X 0.033,Y -490.046,Z 231.000,A 0.000,B 0.000,C 90.000,E1 52.029} C_DIS
LIN {X -0.125,Y -490.718,Z 231.000,A 0.000,B 0.000,C 90.000,E1 51.743} C_DIS
LIN {X 0.101,Y -491.118,Z 231.000,A 0.000,B 0.000,C 90.000,E1 51.412} C_DIS
LIN {X 0.175,Y -491.162,Z 231.000,A 0.000,B 0.000,C 90.000,E1 51.251} C_DIS
LIN {X 0.251,Y -491.618,Z 231.000,A 0.000,B 0.000,C 90.000,E1 51.090} C_DIS
LIN {X 0.096,Y -492.315,Z 231.000,A 0.000,B 0.000,C 90.000,E1 50.803} C_DIS
LIN {X 0.102,Y -493.329,Z 231.000,A 0.000,B 0.000,C 90.000,E1 50.194} C_DIS
LIN {X -0.050,Y -493.535,Z 231.000,A 0.000,B 0.000,C 90.000,E1 49.908} C_DIS
LIN {X 0.077,Y -493.290,Z 231.000,A 0.000,B 0.000,C 90.000,E1 49.666} C_DIS
LIN {X -0.031,Y -494.636,Z 231.000,A 0.000,B 0.000,C 90.000,E1 49.299} C_DIS
LIN {X -0.183,Y -495.362,Z 231.000,A 0.000,B 0.000,C 90.000,E1 49.013} C_DIS
LIN {X -0.006,Y -495.808,Z 231.000,A 0.000,B 0.000,C 90.000,E1 48.690} C_DIS
LIN {X -0.153,Y -495.562,Z 231.000,A 0.000,B 0.000,C 90.000,E1 48.405} C_DIS
LIN {X 0.311,Y -494.869,Z 231.000,A 0.000,B 0.000,C 90.000,E1 48.162} C_DIS
LIN {X 0.270,Y -494.863,Z 231.000,A 0.000,B 0.000,C 90.000,E1 48.162} C_DIS
LIN {X 0.031,Y -495.342,Z 231.000,A 0.000,B 0.000,C 90.000,E1 48.081} C_DIS
LIN {X 0.062,Y -496.573,Z 231.000,A 0.000,B 0.000,C 90.000,E1 47.472} C_DIS
LIN {X 0.249,Y -496.869,Z 231.000,A 0.000,B 0.000,C 90.000,E1 47.148} C_DIS
LIN {X -0.071,Y -498.042,Z 231.000,A 0.000,B 0.000,C 90.000,E1 46.581} C_DIS
LIN {X -0.219,Y -498.493,Z 231.000,A 0.000,B 0.000,C 90.000,E1 46.296} C_DIS
LIN {X -0.023,Y -498.215,Z 231.000,A 0.000,B 0.000,C 90.000,E1 45.972} C_DIS
LIN {X -0.292,Y -497.364,Z 231.000,A 0.000,B 0.000,C 90.000,E1 45.810} C_DIS
LIN {X 0.024,Y -497.340,Z 231.000,A 0.000,B 0.000,C 90.000,E1 45.769} C_DIS
LIN {X 0.176,Y -498.111,Z 231.000,A 0.000,B 0.000,C 90.000,E1 45.648} C_DIS
LIN {X 0.021,Y -499.160,Z 231.000,A 0.000,B 0.000,C 90.000,E1 45.364} C_DIS
LIN {X -0.136,Y -499.262,Z 231.000,A 0.000,B 0.000,C 90.000,E1 45.081} C_DIS
LIN {X 0.067,Y -498.477,Z 231.000,A 0.000,B 0.000,C 90.000,E1 44.757} C_DIS
LIN {X 0.117,Y -498.041,Z 231.000,A 0.000,B 0.000,C 90.000,E1 44.676} C_DIS
LIN {X 0.076,Y -498.042,Z 231.000,A 0.000,B 0.000,C 90.000,E1 44.676} C_DIS
LIN {X 0.168,Y -498.394,Z 231.000,A 0.000,B 0.000,C 90.000,E1 44.595} C_DIS
LIN {X 0.269,Y -498.849,Z 231.000,A 0.000,B 0.000,C 90.000,E1 44.433} C_DIS
LIN {X -0.237,Y -499.095,Z 231.000,A 0.000,B 0.000,C 90.000,E1 44.190} C_DIS
LIN {X -0.037,Y -498.699,Z 231.000,A 0.000,B 0.000,C 90.000,E1 43.866} C_DIS
LIN {X 0.176,Y -498.487,Z 231.000,A 0.000,B 0.000,C 90.000,E1 43.785} C_DIS
LIN {X 0.135,Y -498.504,Z 231.000,A 0.000,B 0.000,C 90.000,E1 43.785} C_DIS
LIN {X 0.063,Y -499.021,Z 231.000,A 0.000,B 0.000,C 90.000,E1 43.704} C_DIS
LIN {X 0.163,Y -499.550,Z 231.000,A 0.000,B 0.000,C 90.000,E1 43.542} C_DIS
LIN {X 0.020,Y -499.845,Z 231.000,A 0.000,B 0.000,C 90.000,E1 43.257} C_DIS
LIN {X 0.223,Y -499.675,Z 231.000,A 0.000,B 0.000,C 90.000,E1 42.933} C_DIS
LIN {X -0.166,Y -498.963,Z 231.000,A 0.000,B 0.000,C 90.000,E1 42.771} C_DIS
LIN {X -0.248,Y -498.912,Z 231.000,A 0.000,B 0.000,C 90.000,E1 42.771} C_DIS
LIN {X -0.289,Y -498.904,Z 231.000,A 0.000,B 0.000,C 90.000,E1 42.771} C_DIS
LIN {X -0.280,Y -499.276,Z 231.000,A 0.000,B 0.000,C 90.000,E1 42.690} C_DIS
LIN {X -0.081,Y -499.867,Z 231.000,A 0.000,B 0.000,C 90.000,E1 42.366} C_DIS
LIN {X -0.218,Y -499.730,Z 231.000,A 0.000,B 0.000,C 90.000,E1 42.081} C_DIS
LIN {X -0.180,Y -498.448,Z 231.000,A 0.000,B 0.000,C 90.000,E1 41.757} C_DIS
LIN {X -0.303,Y -498.350,Z 231.000,A 0.000,B 0.000,C 90.000,E1 41.757} C_DIS
LIN {X 0.028,Y -498.360,Z 231.000,A 0.000,B 0.000,C 90.000,E1 41.714} C_DIS
LIN {X 0.082,Y -498.952,Z 231.000,A 0.000,B 0.000,C 90.000,E1 41.595} C_DIS
LIN {X -0.150,Y -499.408,Z 231.000,A 0.000,B 0.000,C 90.000,E1 41.472} C_DIS
LIN {X 0.047,Y -499.526,Z 231.000,A 0.000,B 0.000,C 90.000,E1 41.148} C_DIS
LIN {X -0.035,Y -498.182,Z 231.000,A 0.000,B 0.000,C 90.000,E1 40.782} C_DIS
LIN {X 0.136,Y -497.917,Z 231.000,A 0.000,B 0.000,C 90.000,E1 40.701} C_DIS
LIN {X 0.095,Y -497.899,Z 231.000,A 0.000,B 0.000,C 90.000,E1 40.701} C_DIS
LIN {X 0.111,Y -498.357,Z 231.000,A 0.000,B 0.000,C 90.000,E1 40.539} C_DIS
LIN {X -0.024,Y -498.908,Z 231.000,A 0.000,B 0.000,C 90.000,E1 40.253} C_DIS
LIN {X 0.034,Y -498.544,Z 231.000,A 0.000,B 0.000,C 90.000,E1 39.644} C_DIS
LIN {X -0.042,Y -497.881,Z 231.000,A 0.000,B 0.000,C 90.000,E1 38.749} C_DIS
LIN {X -0.303,Y -497.180,Z 231.000,A 0.000,B 0.000,C 90.000,E1 38.177} C_DIS
LIN {X 0.262,Y -496.669,Z 231.000,A 0.000,B 0.000,C 90.000,E1 37.810} C_DIS
LIN {X 0.130,Y -496.416,Z 231.000,A 0.000,B 0.000,C 90.000,E1 37.523} C_DIS
LIN {X 0.278,Y -494.749,Z 231.000,A 0.000,B 0.000,C 90.000,E1 36.297} C_DIS
LIN {X -0.038,Y -492.319,Z 231.000,A 0.000,B 0.000,C 90.000,E1 34.818} C_DIS
LIN {X 0.066,Y -491.326,Z 231.000,A 0.000,B 0.000,C 90.000,E1 34.199} C_DIS
LIN {X 0.163,Y -490.142,Z 231.000,A 0.000,B 0.000,C 90.000,E1 33.579} C_DIS
LIN {X 0.251,Y -488.863,Z 231.000,A 0.000,B 0.000,C 90.000,E1 32.959} C_DIS
LIN {X 0.137,Y -486.896,Z 231.000,A 0.000,B 0.000,C 90.000,E1 31.750} C_DIS
LIN {X 0.013,Y -485.169,Z 231.000,A 0.000,B 0.000,C 90.000,E1 30.846} C_DIS
LIN {X -0.193,Y -484.487,Z 231.000,A 0.000,B 0.000,C 90.000,E1 30.256} C_DIS
LIN {X 0.039,Y -482.773,Z 231.000,A 0.000,B 0.000,C 90.000,E1 28.999} C_DIS
LIN {X 0.025,Y -482.199,Z 231.000,A 0.000,B 0.000,C 90.000,E1 28.693} C_DIS
LIN {X -0.198,Y -481.546,Z 231.000,A 0.000,B 0.000,C 90.000,E1 28.103} C_DIS
LIN {X 0.112,Y -478.724,Z 231.000,A 0.000,B 0.000,C 90.000,E1 25.283} C_DIS
LIN {X -0.184,Y -477.882,Z 231.000,A 0.000,B 0.000,C 90.000,E1 24.079} C_DIS
LIN {X -0.080,Y -476.751,Z 231.000,A 0.000,B 0.000,C 90.000,E1 22.514} C_DIS
LIN {X 0.211,Y -475.056,Z 231.000,A 0.000,B 0.000,C 90.000,E1 20.301} C_DIS
LIN {X -0.032,Y -474.191,Z 231.000,A 0.000,B 0.000,C 90.000,E1 19.396} C_DIS
LIN {X -0.093,Y -473.882,Z 231.000,A 0.000,B 0.000,C 90.000,E1 18.779} C_DIS
LIN {X -0.120,Y -472.737,Z 231.000,A 0.000,B 0.000,C 90.000,E1 17.221} C_DIS
LIN {X 0.111,Y -471.960,Z 231.000,A 0.000,B 0.000,C 90.000,E1 16.567} C_DIS
LIN {X 0.109,Y -471.471,Z 231.000,A 0.000,B 0.000,C 90.000,E1 15.315} C_DIS
LIN {X 0.124,Y -470.158,Z 231.000,A 0.000,B 0.000,C 90.000,E1 13.119} C_DIS
LIN {X 0.061,Y -469.168,Z 231.000,A 0.000,B 0.000,C 90.000,E1 11.243} C_DIS
LIN {X -0.209,Y -468.827,Z 231.000,A 0.000,B 0.000,C 90.000,E1 10.018} C_DIS
LIN {X -0.198,Y -468.126,Z 231.000,A 0.000,B 0.000,C 90.000,E1 7.814} C_DIS
LIN {X -0.098,Y -467.817,Z 231.000,A 0.000,B 0.000,C 90.000,E1 6.543} C_DIS
LIN {X -0.010,Y -467.755,Z 231.000,A 0.000,B 0.000,C 90.000,E1 2.751} C_DIS
LIN {X 0.000,Y -468.333,Z 231.000,A 0.000,B 0.000,C 90.000,E1 360.000} C_DIS
LIN {X 0.000,Y -593.333,Z 231.000,A 0.000,B 0.000,C 89.370,E1 360.000} C_DIS
SetRpm(0)

END
